(* IEC 61131-3 sources: factoryforge/examples/graded, 1 file *)

(* ---- first_hour_sorting_by_height.st ---- *)
(* ------------------------------------------------------------------------
   FactoryForge starter -- Sorting by height (scene sorting-by-height)
   OpenPLC Runtime v3, IEC 61131-3 Structured Text, over Modbus TCP.
   Generated by tools/gen_starters.py from the scene's tag set; see README.md
   beside this file. Write your program in section 2 below.

   THE TASK
     Run the belt, feed cartons, and push the tall ones down the chute
     while the short ones carry on. Two sensors at two heights are all you
     get: a carton that breaks the high beam is tall, one that breaks only
     the low beam is short.

   DONE WHEN
     Every tall carton ends up in the chute and every short one at the far
     end, with counter.tall and counter.short adding up to what you fed.
     The mushroom stops the line inside 200 ms and Start alone will not
     restart it. If the belt's drive faults (conveyor.fault), stop feeding,
     and when the fault clears stay stopped until Reset, then Start.

     NOTE: This is the line the 3D engine opens and the grader marks:
     nineteen tags, with an operator panel and two fault contacts.
     `factoryforge-sidecar demo` runs a different, ten-tag Python scene
     whose Modbus map is NOT this one; the finished program for that one is
     examples/openplc/Sorting.st.

   HOW IT IS WIRED
     FactoryForge is the Modbus slave; OpenPLC is the master and polls it.
     mbconfig.cfg beside this file is that Slave Device. The addresses
     below are the ones the sidecar serves for this scene when it is
     started AFTER the scene is open, in the folder FactoryForge was
     extracted to:

       .\factoryforge-sidecar connect --driver modbus-tcp -o port 5502

     (./factoryforge-sidecar on Linux.)
     It prints its address map on startup; that map is the authority, and
     the table below must match it line for line. Change scene and the
     sidecar keeps every address it has handed out and puts new tags above
     them -- restart it after changing scene.

     OpenPLC numbers each block it polls from 100: slave coil n is
     %QX(100 + n/8).(n mod 8), slave input register n is %IW(100 + n).

     An INT or REAL tag is 32 bits and takes TWO registers, high word
     first. Section 1 rebuilds the inputs and section 3 splits the outputs;
     your program works with the plain DINT and REAL variables.

     In the sidecar's order (block, then address; addresses are decimal):

     MODBUS   REGS  OPENPLC                TAG
     0x0      1     %QX100.0               conveyor.rotate
     0x1      1     %QX100.1               emitter.emit
     0x2      1     %QX100.2               panel.green
     0x3      1     %QX100.3               panel.red
     0x4      1     %QX100.4               pusher.extend
     0x5      1     %QX100.5               stack_light.green
     1x0      1     %IX100.0               conveyor.fault
     1x1      1     %IX100.1               panel.estop
     1x2      1     %IX100.2               panel.reset
     1x3      1     %IX100.3               panel.start
     1x4      1     %IX100.4               panel.stop
     1x5      1     %IX100.5               pusher.extended
     1x6      1     %IX100.6               pusher.fault
     1x7      1     %IX100.7               pusher.retracted
     1x8      1     %IX101.0               sensor_high.detect
     1x9      1     %IX101.1               sensor_low.detect
     3x0      2     %IW100 + %IW101        counter.short
     3x2      2     %IW102 + %IW103        counter.tall
     3x4      2     %IW104 + %IW105        panel.setpoint
   ------------------------------------------------------------------------ *)

(* The sidecar sends a 32-bit value as two registers, high word first
   (struct.pack(">i") in drivers/modbus_tcp.py). DWORD_TO_DINT reinterprets
   the bit pattern, so this is right for negative values too. *)
FUNCTION FF_WORDS_TO_DINT : DINT
  VAR_INPUT
    HI : WORD;
    LO : WORD;
  END_VAR
  FF_WORDS_TO_DINT := DWORD_TO_DINT(SHL(IN := WORD_TO_DWORD(HI), N := 16)
                                    OR WORD_TO_DWORD(LO));
END_FUNCTION

(* A REAL arrives the same way: IEEE-754 single precision, high word first.
   OpenPLC's DWORD_TO_REAL cannot rebuild it -- it converts the NUMBER, so
   16#3F800000 becomes 1065353216.0 rather than 1.0 -- so this takes the
   sign, exponent and mantissa apart by hand. Exact for every normal value;
   zero and the tiny subnormals (below 1.2E-38) come back as 0.0. *)
FUNCTION FF_WORDS_TO_REAL : REAL
  VAR_INPUT
    HI : WORD;
    LO : WORD;
  END_VAR
  VAR
    Exponent : INT;
    Value    : REAL;
  END_VAR
  Exponent := WORD_TO_INT(SHR(IN := HI, N := 7) AND 16#00FF);
  IF Exponent = 0 OR Exponent = 255 THEN
    Value := 0.0;
  ELSE
    Value := 1.0 + DWORD_TO_REAL(SHL(IN := WORD_TO_DWORD(HI AND 16#007F), N := 16)
                                 OR WORD_TO_DWORD(LO)) / 8388608.0;
    Exponent := Exponent - 127;
    WHILE Exponent > 0 DO
      Value := Value * 2.0;
      Exponent := Exponent - 1;
    END_WHILE;
    WHILE Exponent < 0 DO
      Value := Value / 2.0;
      Exponent := Exponent + 1;
    END_WHILE;
    IF (HI AND 16#8000) <> 0 THEN
      Value := -Value;
    END_IF;
  END_IF;
  FF_WORDS_TO_REAL := Value;
END_FUNCTION

PROGRAM sorting_by_height
  VAR
    (* --- PLC writes: coils --------------------------------------------- *)
    ConveyorRotate  AT %QX100.0  : BOOL;  (* conveyor.rotate   0x0   run the belt *)
    EmitterEmit     AT %QX100.1  : BOOL;  (* emitter.emit      0x1   rising edge = feed one carton; hold each level well over one poll *)
    PanelGreen      AT %QX100.2  : BOOL;  (* panel.green       0x2   green lamp on the panel *)
    PanelRed        AT %QX100.3  : BOOL;  (* panel.red         0x3   red lamp on the panel *)
    PusherExtend    AT %QX100.4  : BOOL;  (* pusher.extend     0x4   extend the pusher *)
    StackLightGreen AT %QX100.5  : BOOL;  (* stack_light.green 0x5   green tower lamp *)
    (* --- PLC reads: discrete inputs ------------------------------------ *)
    ConveyorFault    AT %IX100.0  : BOOL;  (* conveyor.fault     1x0   drive fault: TRUE = faulted; a faulted drive does not turn, whatever it is told *)
    PanelEstop       AT %IX100.1  : BOOL;  (* panel.estop        1x1   E-stop, normally closed: TRUE = healthy, FALSE = pressed; stays pressed until pulled out *)
    PanelReset       AT %IX100.2  : BOOL;  (* panel.reset        1x2   Reset button, momentary: a short pulse per press *)
    PanelStart       AT %IX100.3  : BOOL;  (* panel.start        1x3   Start button, momentary: a short pulse per press -- latch it *)
    PanelStop        AT %IX100.4  : BOOL;  (* panel.stop         1x4   Stop button, momentary: a short pulse per press *)
    PusherExtended   AT %IX100.5  : BOOL;  (* pusher.extended    1x5   pusher fully out *)
    PusherFault      AT %IX100.6  : BOOL;  (* pusher.fault       1x6   drive fault: TRUE = jammed; it freezes where it is *)
    PusherRetracted  AT %IX100.7  : BOOL;  (* pusher.retracted   1x7   pusher fully back *)
    SensorHighDetect AT %IX101.0  : BOOL;  (* sensor_high.detect 1x8   high beam: TRUE while a TALL carton is in it *)
    SensorLowDetect  AT %IX101.1  : BOOL;  (* sensor_low.detect  1x9   low beam: TRUE while any carton is in it *)
    (* --- PLC reads: input registers, two per value --------------------- *)
    CounterShortHi  AT %IW100    : WORD;  (* counter.short  3x0   high word of CounterShort *)
    CounterShortLo  AT %IW101    : WORD;  (* counter.short  3x1   low word of CounterShort *)
    CounterTallHi   AT %IW102    : WORD;  (* counter.tall   3x2   high word of CounterTall *)
    CounterTallLo   AT %IW103    : WORD;  (* counter.tall   3x3   low word of CounterTall *)
    PanelSetpointHi AT %IW104    : WORD;  (* panel.setpoint 3x4   high word of PanelSetpoint *)
    PanelSetpointLo AT %IW105    : WORD;  (* panel.setpoint 3x5   low word of PanelSetpoint *)
  END_VAR

  (* A second VAR block, and not for tidiness: matiec will not mix located
     and unlocated declarations in one. Your own variables go here too. *)
  VAR
    (* --- PLC reads, in engineering units ---------------------------------- *)
    CounterShort  : DINT;  (* counter.short  cartons that reached the end of the belt, running total *)
    CounterTall   : DINT;  (* counter.tall   cartons that came down the chute, running total *)
    PanelSetpoint : REAL;  (* panel.setpoint the operator's pot, 0.3..1.8 s (starts at 0.9) *)
    Running   : BOOL;    (* the line is running *)
    Tripped   : BOOL;    (* the E-stop or a drive fault tripped; only Reset clears it *)
    EstopSeen : BOOL;    (* the E-stop has read healthy since OpenPLC started *)
    rStart    : R_TRIG;  (* the moment Start goes down *)
    rReset    : R_TRIG;  (* the moment Reset goes down *)
    tEmit     : TON;     (* times the feed: one carton every 3 s *)
    EmitFlag  : BOOL;
    HighMem   : BOOL;    (* the high beam, one scan ago *)
    PushReq   : BOOL;    (* a tall carton is on its way to the pusher *)
    tDelay    : TON;     (* high beam -> carton in front of the pusher *)
    tPush     : TON;     (* how long the pusher stays out *)
  END_VAR

  (* ===== 1. Inputs: rebuild each 32-bit value from its two registers ===== *)
  CounterShort := FF_WORDS_TO_DINT(HI := CounterShortHi, LO := CounterShortLo);
  CounterTall := FF_WORDS_TO_DINT(HI := CounterTallHi, LO := CounterTallLo);
  PanelSetpoint := FF_WORDS_TO_REAL(HI := PanelSetpointHi, LO := PanelSetpointLo);

  (* ===== 2. Your program ================================================
     The task is at the top of this file and in the scene's Task panel.
     Every signal above can be used by name here: the bits directly, the
     32-bit values through CounterShort, CounterTall, PanelSetpoint.

     FIRST SCANS READ FALSE. OpenPLC scans before its first Modbus poll
     returns, and until then every input reads FALSE. PanelEstop is
     normally closed, so it looks struck, and a trip latched on NOT
     PanelEstop trips itself every time OpenPLC starts. Arm the trip
     only once the E-stop has read healthy, and keep refusing Start
     while it reads FALSE (docs/OPENPLC.md, Troubleshooting):
       EstopSeen : BOOL;   in the second VAR block
       IF PanelEstop THEN EstopSeen := TRUE; END_IF;
       IF EstopSeen AND NOT PanelEstop THEN Tripped := TRUE; END_IF; *)

  (* The operator panel. Start and Reset are momentary: act on the scan
     the button goes down, not for as long as it is held. *)
  rStart(CLK := PanelStart);
  rReset(CLK := PanelReset);

  (* Until OpenPLC's first poll reaches the slave, every input reads
     FALSE, and a normally closed E-stop that reads FALSE looks struck.
     So a trip only counts once the E-stop has been seen healthy. *)
  IF PanelEstop THEN
    EstopSeen := TRUE;
  END_IF;

  (* The E-stop trips the line, and so does the belt's drive faulting.
     The trip latches: releasing the mushroom or the fault clearing does
     not clear it, and neither does Start. Only Reset does, and not while
     the fault is still there. *)
  IF (EstopSeen AND NOT PanelEstop) OR ConveyorFault THEN
    Tripped := TRUE;
  ELSIF rReset.Q THEN
    Tripped := FALSE;
  END_IF;

  (* Start runs the line, and only while the E-stop reads healthy. Stop or
     a trip stops it. Reset alone does not start anything: after a trip it
     takes Reset, then Start. *)
  IF Tripped OR PanelStop OR NOT PanelEstop THEN
    Running := FALSE;
  ELSIF rStart.Q THEN
    Running := TRUE;
  END_IF;

  ConveyorRotate  := Running;
  StackLightGreen := Running;
  PanelGreen      := Running;
  PanelRed        := Tripped;

  (* Feed while the line runs: a square wave, 1.5 s high and 1.5 s low,
     one carton per rising edge. A short pulse would be missed: OpenPLC
     polls every 50 ms. *)
  IF Running THEN
    tEmit(IN := TRUE, PT := T#1500ms);
    IF tEmit.Q THEN
      EmitFlag := NOT EmitFlag;
      tEmit(IN := FALSE, PT := T#1500ms);
    END_IF;
  ELSE
    tEmit(IN := FALSE, PT := T#1500ms);
    EmitFlag := FALSE;
  END_IF;
  EmitterEmit := EmitFlag;

  (* A tall carton breaks the high beam 1.2 s before it reaches the pusher,
     and the pusher takes 0.3 s to come out: wait 0.9 s, then push. *)
  IF SensorHighDetect AND NOT HighMem THEN
    PushReq := TRUE;
  END_IF;
  HighMem := SensorHighDetect;
  tDelay(IN := PushReq, PT := T#900ms);
  tPush(IN := tDelay.Q, PT := T#1500ms);
  PusherExtend := tDelay.Q AND NOT tPush.Q;
  IF tPush.Q THEN
    PushReq := FALSE;
  END_IF;

  (* ===== 3. Outputs: split each 32-bit value into its two registers ===== *)
  (* none in this scene *)

END_PROGRAM

CONFIGURATION Config0

  RESOURCE Res0 ON PLC
    (* 20 ms, as in examples/openplc/Sorting.st: every scan spent waiting
       comes out of the scene's timing margins. *)
    TASK Main(INTERVAL := T#20ms, PRIORITY := 0);
    PROGRAM Inst0 WITH Main : sorting_by_height;
  END_RESOURCE

END_CONFIGURATION
